{attribute addProperty BoxType "EL1259-0000-0017"}
{attribute addProperty Id "Output_buffer_resetBIT10.1251Manual_output_stateBIT10.1252Force_orderBIT10.1253Enable_manual_operationBIT10.1254Output_order_counterUSINT819No_of_output_eventsUSINT8117"}
{attribute addProperty CRC "2397020335"}
{attribute addProperty SizeInBites "60"}
{attribute addProperty SizeInBytes "7.5"}
{warning 'Size of this structure is not a multiple of 8 bits!!!'}
TYPE Ctrl_8EDFA0AF :
STRUCT
	{attribute addProperty Name "Output_buffer_reset"}
	Output_buffer_reset : BIT;
	{attribute addProperty Name "Manual_output_state"}
	Manual_output_state : BIT;
	{attribute addProperty Name "Force_order"}
	Force_order : BIT;
	{attribute addProperty Name "Enable_manual_operation"}
	Enable_manual_operation : BIT;
	{attribute 'hide'}
	reserve_1_BOOL_0 : BOOL;
	{attribute 'hide'}
	reserve_1_BOOL_1 : BOOL;
	{attribute 'hide'}
	reserve_1_BOOL_2 : BOOL;
	{attribute 'hide'}
	reserve_1_BOOL_3 : BOOL;
	{attribute addProperty Name "Output_order_counter"}
	Output_order_counter : USINT;
	{attribute addProperty Name "No_of_output_events"}
	No_of_output_events : USINT;
	{attribute 'hide'}
	reserve_2 : BYTE;
END_STRUCT
END_TYPE

(* stored: Version 1.2.0.0, ProductVersion 3.1.4024.9
   DUT Ctrl_8EDFA0AF: Id {6d2d3b62-c799-4f53-afc4-8d4652f51b2d} *)
